{attribute 'linkalways'} 
{attribute 'no_explicit_call' := 'This FB is a CLASS and must be accessed using methods or properties'}
{attribute 'enable_dynamic_creation'}
FUNCTION_BLOCK _ETcVnOcrOptions EXTENDS EnumDatatypeBase
VAR
	localData : ETcVnOcrOptions;
	activeData : REFERENCE TO ETcVnOcrOptions;
	enumBaseDatatype : _UDINT(localData);
END_VAR

METHOD PRIVATE AddLocalEnumeration
VAR_INPUT
	Enumeration : T_MAXSTRING;
	Value : ETcVnOcrOptions;
END_VAR
AddEnumeration(Enumeration, Value);
END_METHOD

PROPERTY PUBLIC Address : PVOID
GET
Address := ADR(activeData);
END_GET
END_PROPERTY

METHOD PUBLIC ClearReference
VAR_INPUT
END_VAR
activeData REF= localData;
SetBaseDatatypeReference();
END_METHOD

METHOD PUBLIC Clone : I_Datatype
VAR
    pClone : POINTER TO _ETcVnOcrOptions;
END_VAR
pClone := __NEW(_ETcVnOcrOptions(InitialValue := Value));
Clone := pClone^;
END_METHOD

METHOD FB_init : BOOL
VAR_INPUT
	bInitRetains : BOOL; // if TRUE, the retain variables are initialized (warm start / cold start)
	bInCopyCode : BOOL;  // if TRUE, the instance afterwards gets moved into the copy code (online change)
	InitialValue : ETcVnOcrOptions;
END_VAR
localData := InitialValue;
AddBaseDatatype(enumBaseDatatype);
ClearReference();

AddLocalEnumeration('TCVN_OO_WITHBLANKS', ETcVnOcrOptions.TCVN_OO_WITHBLANKS);
END_METHOD

PROPERTY PUBLIC Identifier : T_MAXSTRING
GET
Identifier := 'ETcVnOcrOptions';
END_GET
END_PROPERTY

METHOD IsEnumeratorValueEqual : BOOL
VAR_INPUT
	Enumerator : I_KeyValueForwardEnumerator;
END_VAR
VAR
	storedValue : ETcVnOcrOptions;
END_VAR
IF NOT Enumerator.TryGet(storedValue) THEN
	RETURN;
END_IF

IsEnumeratorValueEqual := storedValue = activeData;
END_METHOD

METHOD PUBLIC MakeReferenceTo
VAR_INPUT
	ReferenceTarget : REFERENCE TO ETcVnOcrOptions;
END_VAR
activeData REF= ReferenceTarget;
SetBaseDatatypeReference();
END_METHOD

METHOD PROTECTED SetBaseDatatypeReference
VAR_INPUT
END_VAR
enumBaseDatatype.MakeReferenceTo(activeData);
END_METHOD

PROPERTY PUBLIC Size : UDINT
GET
Size := SIZEOF(activeData);
END_GET
END_PROPERTY

METHOD TryMakeReferenceTo : BOOL
VAR_INPUT
	Target : I_Datatype;
END_VAR
VAR
	targetAsEnum : I_EnumDatatype;
	pTargetData : POINTER TO ETcVnOcrOptions;
END_VAR
IF NOT Target.TryResolveAsEnumDatatype(targetAsEnum) THEN
	RETURN;
END_IF

IF targetAsEnum.Identifier <> Identifier THEN
	RETURN;
END_IF

pTargetData := Target.Address;
activeData REF= pTargetData^;
SetBaseDatatypeReference();
TryMakeReferenceTo := TRUE;
END_METHOD

PROPERTY PUBLIC Value : ETcVnOcrOptions
GET
Value := activeData;
END_GET
SET
activeData := Value;
END_SET
END_PROPERTY

END_FUNCTION_BLOCK

(* stored: Version 1.1.0.1, ProductVersion 3.1.4024.12
   POU _ETcVnOcrOptions: Id {58936afd-3ec5-44d5-8db3-4019bd138e8c}, SpecialFunc None
   Folder Constructor: Id {f58f565a-f860-4c02-8c74-e49aeafad45a}
   Folder Private: Id {d8de498b-7c91-4b3c-b208-7e80b9341fe0}
   Folder Protected: Id {c55d1630-10f8-4118-9fd1-aa192316e7b5}
   Method AddLocalEnumeration: Id {227ba2cc-3b5e-42de-89ea-4250e68bde0b}
   Property Address: Id {560ed570-995b-4fb7-97e9-903c61c9d493}
   Get Get: Id {2722c024-c48e-47b7-8eff-0cd615b5552d}
   Method ClearReference: Id {64b135e7-97f3-4ef2-8fae-e46e85731042}
   Method Clone: Id {43966038-4d61-4860-846f-8a01e6382f9e}
   Method FB_init: Id {16307998-b172-42d2-bfb3-66c988da4b02}
   Property Identifier: Id {c53b4541-39f1-4897-82f1-e1c4ce92e933}
   Get Get: Id {9f56ef32-d899-4f05-9c86-29c86c1431ec}
   Method IsEnumeratorValueEqual: Id {f6085903-4723-4338-904e-698fd9e7bf2f}
   Method MakeReferenceTo: Id {30810507-f978-4040-beff-2acc54b120a5}
   Method SetBaseDatatypeReference: Id {0d5ca6b6-f9b2-4a08-a7b0-2c333bfc0c5e}
   Property Size: Id {b57aecdb-e803-4e60-ae89-17436112d111}
   Get Get: Id {d11c6096-1ec0-4281-8774-40d2b3a9fe94}
   Method TryMakeReferenceTo: Id {cfb5aa0a-5391-4f9c-aad7-09745621ea28}
   Property Value: Id {d8fa8b1b-cfbd-4b0c-9ade-6a48d038d14a}
   Get Get: Id {b85de563-9f2a-4106-bc48-fe89cd9d574d}
   Set Set: Id {32d6427c-0f43-4337-9653-98b96ad6a5d3} *)
